(* IEC 61131-3 sources: Industry-PLC-LLM/data/PLCBEAD_repo/PLCBEAD_PLCEmbed-main/PLC-BEAD/Source/GEB/YEAR_OF_DATE, 1 file *)

(* ---- YEAR_OF_DATE.ST ---- *)
FUNCTION YEAR_OF_DATE:INT
	VAR_INPUT
		IDATE :	UDINT;
	END_VAR

	YEAR_OF_DATE := UDINT_TO_INT((IDATE+UDINT#43200) / UDINT#31557600 + UDINT#1970);
END_FUNCTION

PROGRAM program0
  VAR
    LocalVar0 : UDINT;
    CEIL5_OUT : INT;
  END_VAR

  CEIL5_OUT := YEAR_OF_DATE(LocalVar0);
END_PROGRAM
